TYPE u_LedColor :
UNION
	dw_LedColor	:	DWORD;
	st_LedColor	:	st_LedColor;
END_UNION
END_TYPE

(* stored: Version 1.1.0.1, ProductVersion 3.1.4024.12
   DUT u_LedColor: Id {4cc238ce-a0d4-40c9-9910-7e0e92d57190} *)
